Fanuc KAREL source: IO0197.KL

-- PROVISIONAL review KL for V770-1; original PC SHA256 c279a5df81e9e81c9238d338bc3b109232003549b388795e1f96dfe869f15311
-- Incomplete behavior may be omitted. Consult companion uncertainty JSON. Do not deploy.
PROGRAM IO0197
%NOLOCKGROUP
-- UNRESOLVED_LOCAL_POOL 5 cells at code offset 13; source declarations unknown
-- DIRECT_LOCAL_WORD_ACCESS alone does not prove INTEGER, REAL, or BOOLEAN
BEGIN
  -- UNRESOLVED_PC offsets 0-18; opcodes 2B,2C,7B
  -- UNRESOLVED_PC offsets 23-30; opcodes 9D,23
  -- UNRESOLVED_PC offsets 35-49; opcodes 2E,22,9D,33,35
  -- UNRESOLVED_PC offsets 54-61; opcodes 9D,23
  -- UNRESOLVED_PC offsets 66-77; opcodes 2E,23
  -- UNRESOLVED_PC offsets 82-108; opcodes 27,27,9D,22,27,9D,31,7E,4A
  -- UNRESOLVED_PC offsets 113-117; opcodes 7F
  -- UNRESOLVED_PC offsets 122-126; opcodes 27,AA
  -- UNRESOLVED_PC offsets 131-135; opcodes 7F
END IO0197
